{attribute 'qualified_only'}
{attribute 'strict'}
{attribute 'to_string'}
TYPE E_JOB_CHECK :
(
  CHECK_NULL,

  POINTER_NULL                        :=  9000,
  POINTER_NULL_UNIT_CTRL,
  POINTER_NULL_UNIT_STATE,

  POINTER_NULL_AXIS_CTRL              :=  9010,
  POINTER_NULL_AXIS_STATE,
  POINTER_NULL_AXIS_INFO,
  POINTER_NULL_AXIS_MOVE_DATA,
  POINTER_NULL_AXIS_INDEX,
  POINTER_NULL_AXIS_IDENTITY,

  POINTER_NULL_NCI_CHN_CTRL           :=  9020,
  POINTER_NULL_NCI_CHN_STATE,

  POINTER_NULL_JOB_PARAMETER          :=  9030,

  POINTER_NULL_SCALE_COM_CONTROL      :=  9040,
  POINTER_NULL_SCALE_COM_STATE,
  POINTER_NULL_SCALE_CONFIG,

  AXIS_RANGE_START_INVALID            :=  9100,
  AXIS_RANGE_END_INVALID,
  AXIS_DISPENSER_COMPONENTS_INVALID,

  NCI_CONFIGURATION_INVALID           :=  9200,
  CHANNEL_INDEX_INVALID,
  NCI_R_PARAMETER_INVALID,
  NCI_FILE_CTRL_INVALID,
  NCI_FILE_STATE_INVALID,

  POINTER_NULL_HOME_PARAMETER         :=  9300,
  POINTER_NULL_RINSE_PARAMETER,
  POINTER_NULL_WEIGH_PARAMETER,
  POINTER_NULL_MEAS_PARAMETER,
  POINTER_NULL_AUTO_PARAMETER,
  POINTER_NULL_STRIP_PARAMETER,

  POINTER_NULL_DISPENSER_PARAMETER    :=  9310,

  INTERFACE_NULL                      :=  9900,
  INTERFACE_NULL_UNIT_CTRL,
  INTERFACE_NULL_DISPENSER,

  CHECK_DONE                          := 10000

)UINT;
END_TYPE

(* stored: Version 1.1.0.1
   DUT E_JOB_CHECK: Id {cf36c09d-0150-075e-3ac1-481c2f4916f5} *)
